Staubli VAL3: checkIn.pgx

program checkIn(string x_sItem (dimensions=1), bool& x_bResult[] (dimensions=1))
  local bool l_bMode[3]
  local string l_sItem[3]
  local num l_nCount
  local num l_nFlag
  local bool l_bActive
  local bool l_bFound
  local num l_nSize
  local num i
  local num j
  local string l_sName
  local string l_sMode
  local bool l_bStatus[3]
begin
  x_bResult=false
  //
  // find how many time and fill sItem and l_bMode
  //
  l_nCount=-1
  do
    l_nCount=l_nCount+1
    // l_sMode
    i=find(x_sItem,"AND")
    if i==-1
      i=find(x_sItem,"OR")
      if i!=-1
        l_sMode="OR"
        i=i+len("OR")+1
      endIf
    else
      l_sMode="AND"
      i=i+len("AND")+1
    endIf
    //
    if i!=-1
      l_sItem[l_nCount]=left(x_sItem,i)
      x_sItem=right(x_sItem,len(x_sItem)-i)
    else
      l_sItem[l_nCount]=x_sItem
    endIf
    l_nFlag=find(l_sItem[l_nCount],">")
    // l_bMode
    if find(l_sItem[l_nCount],">ON")!=-1
      l_bMode[l_nCount]=true
    else
      l_bMode[l_nCount]=false
    endIf
    //sItem
    l_sItem[l_nCount]=left(l_sItem[l_nCount],l_nFlag)
  until i==-1
  //
  call input:getStatus(l_bStatus,l_sItem[0])
  if l_sMode==""
    if (l_bStatus[0]==l_bMode[0])
      x_bResult=true
    endIf
  else
    // more then on event
    call input:getStatus(l_bStatus[1],l_sItem[1])
    //
    if l_sMode=="OR"
      switch l_nCount
        case 1
          if (l_bStatus[0]==l_bMode[0] or l_bStatus[1]==l_bMode[1])
            x_bResult=true
          endIf
        break
        case 2
          call input:getStatus(l_bStatus[2],l_sItem[2])
          if (l_bStatus[0]==l_bMode[0] or l_bStatus[1]==l_bMode[1] or l_bStatus[2]==l_bMode[2])
            x_bResult=true
          endIf
        break
      endSwitch
    else
      if l_sMode=="AND"
        switch l_nCount
          case 1
            if (l_bStatus[0]==l_bMode[0] and l_bStatus[1]==l_bMode[1])
              x_bResult=true
            endIf
          break
          case 2
            call input:getStatus(l_bStatus[2],l_sItem[2])
            if (l_bStatus[0]==l_bMode[0] and l_bStatus[1]==l_bMode[1] and l_bStatus[2]==l_bMode[2])
              x_bResult=true
            endIf
          break
        endSwitch
      endIf
    endIf
  endIf
end
